# EPICS substitutions: db/Beckhoff_5XXX/ecmcEL5072.substitutions
file "ecmcEL5072-chX.template"
{
  pattern {CH_ID}
          {01   }
          {02   }
}
